PROGRAM PressToTargetSim
VAR
	ActPos AT%Q*:	DINT;
	SetVelo AT%I*:	INT;
	PressureA AT%Q*:	INT;
 
 	fSetVelo:	LREAL;
 	fActPos:	LREAL;
	fPressureA:	LREAL;

	bBrake: BOOL;
END_VAR



fSetVelo:=INT_TO_LREAL(SetVelo)/32767*500.0;

fActPos:=fActPos+fSetVelo*0.002;

fActPos:=MIN(MAX(fActPos,0.0),200.0);
ActPos:=LREAL_TO_DINT(fActPos * 1000.0);

fPressureA:=MIN(MAX((fActPos-100.0)*5,0.0),200.0); 

IF bBrake THEN
	fPressureA:=MIN(MAX((fActPos-100.0)*5,0.0),20.0); 
END_IF
PressureA:=LREAL_TO_INT(fPressureA/400.0*32767);

END_PROGRAM

(* stored: Version 1.1.0.1
   POU PressToTargetSim: Id {c34d22a7-9feb-4fd2-a0cd-81eb3ae49bd2}, SpecialFunc None *)
